// TIA Portal V18 export
FUNCTION_BLOCK "ST10_Flow3_A1RotaryShaftScan"   // FB1073, GRAPH
VERSION : 0.1
// stored: AcknowledgeErrorsRequired false, AutoNumber false, GraphVersion 6.0, InitialValuesAcquisition false, IsIECCheckEnabled false, LanguageInNetworks LAD, LockOperatingMode false, PermanentILProcessingInMANMode false, SetENOAutomatically false, SkipSteps false, UDAEnableTagReadback false, WithAlarmHandling true
   // inherited from GRAPH_BASE
   VAR
      OFF_SQ_BASE : Bool;
   END_VAR
   VAR_INPUT
      iSysInface : "RCS_SysComInterface_V1";
   END_VAR
   VAR_IN_OUT
      ioPM_Inface : "RCS_PMInterface_V1";
      ioStatus : Int;
   END_VAR
   VAR
      sCtrlMode { S7_SetPoint := 'True'} : "SysFlowCtrlGraph";
      sUpdMES_Data : Bool;   // 更新MES数据
      工件放行中 : Bool;
      前站站号 { ExternalAccessible := 'False'; ExternalVisible := 'False'; ExternalWritable := 'False'} : UInt;
      本站站号 { ExternalAccessible := 'False'; ExternalVisible := 'False'; ExternalWritable := 'False'} : UInt;
      弹窗Temp : Array[1..10] of Int;
      AlarmID : Int;
      TON { S7_SetPoint := 'True'} : Array[0..10] of TON_TIME;
      TOF { S7_SetPoint := 'True'} : Array[0..10] of TOF_TIME;
      sUP { S7_SetPoint := 'True'} : Array[0..10] of Bool;
      更新RFID完成 : Bool;
   END_VAR
   VAR_TEMP
      Tempresult : USInt;
      本站站号乘10 : UInt;
   END_VAR
   // // TON[0] : 托盘流入1托盘到位传感器 / iA-Rotating product Check
   // // TON[1] : 托盘流入1托盘到位传感器
   // // TON[2] : 托盘流入1产品有无传感器
   // // TON[3] : 托盘流入1产品有无传感器
   // // TON[4] : 托盘流入1姿态检测光电2
   // // TON[5] : 托盘流入1姿态检测光电3
   // // TON[0].Q : 托盘流入1托盘到位 / iA-Rotating product Check
   // // TON[1].Q : 托盘流入1托盘无
   // // TON[2].Q : 托盘流入1有产品
   // // TON[3].Q : 托盘流入1无产品
   // // TON[4].Q : 托盘流入1姿态检测光电2
   // // TON[5].Q : 托盘流入1姿态检测光电3
   // // TOF[1] : iA-Rotating product Check
BEGIN
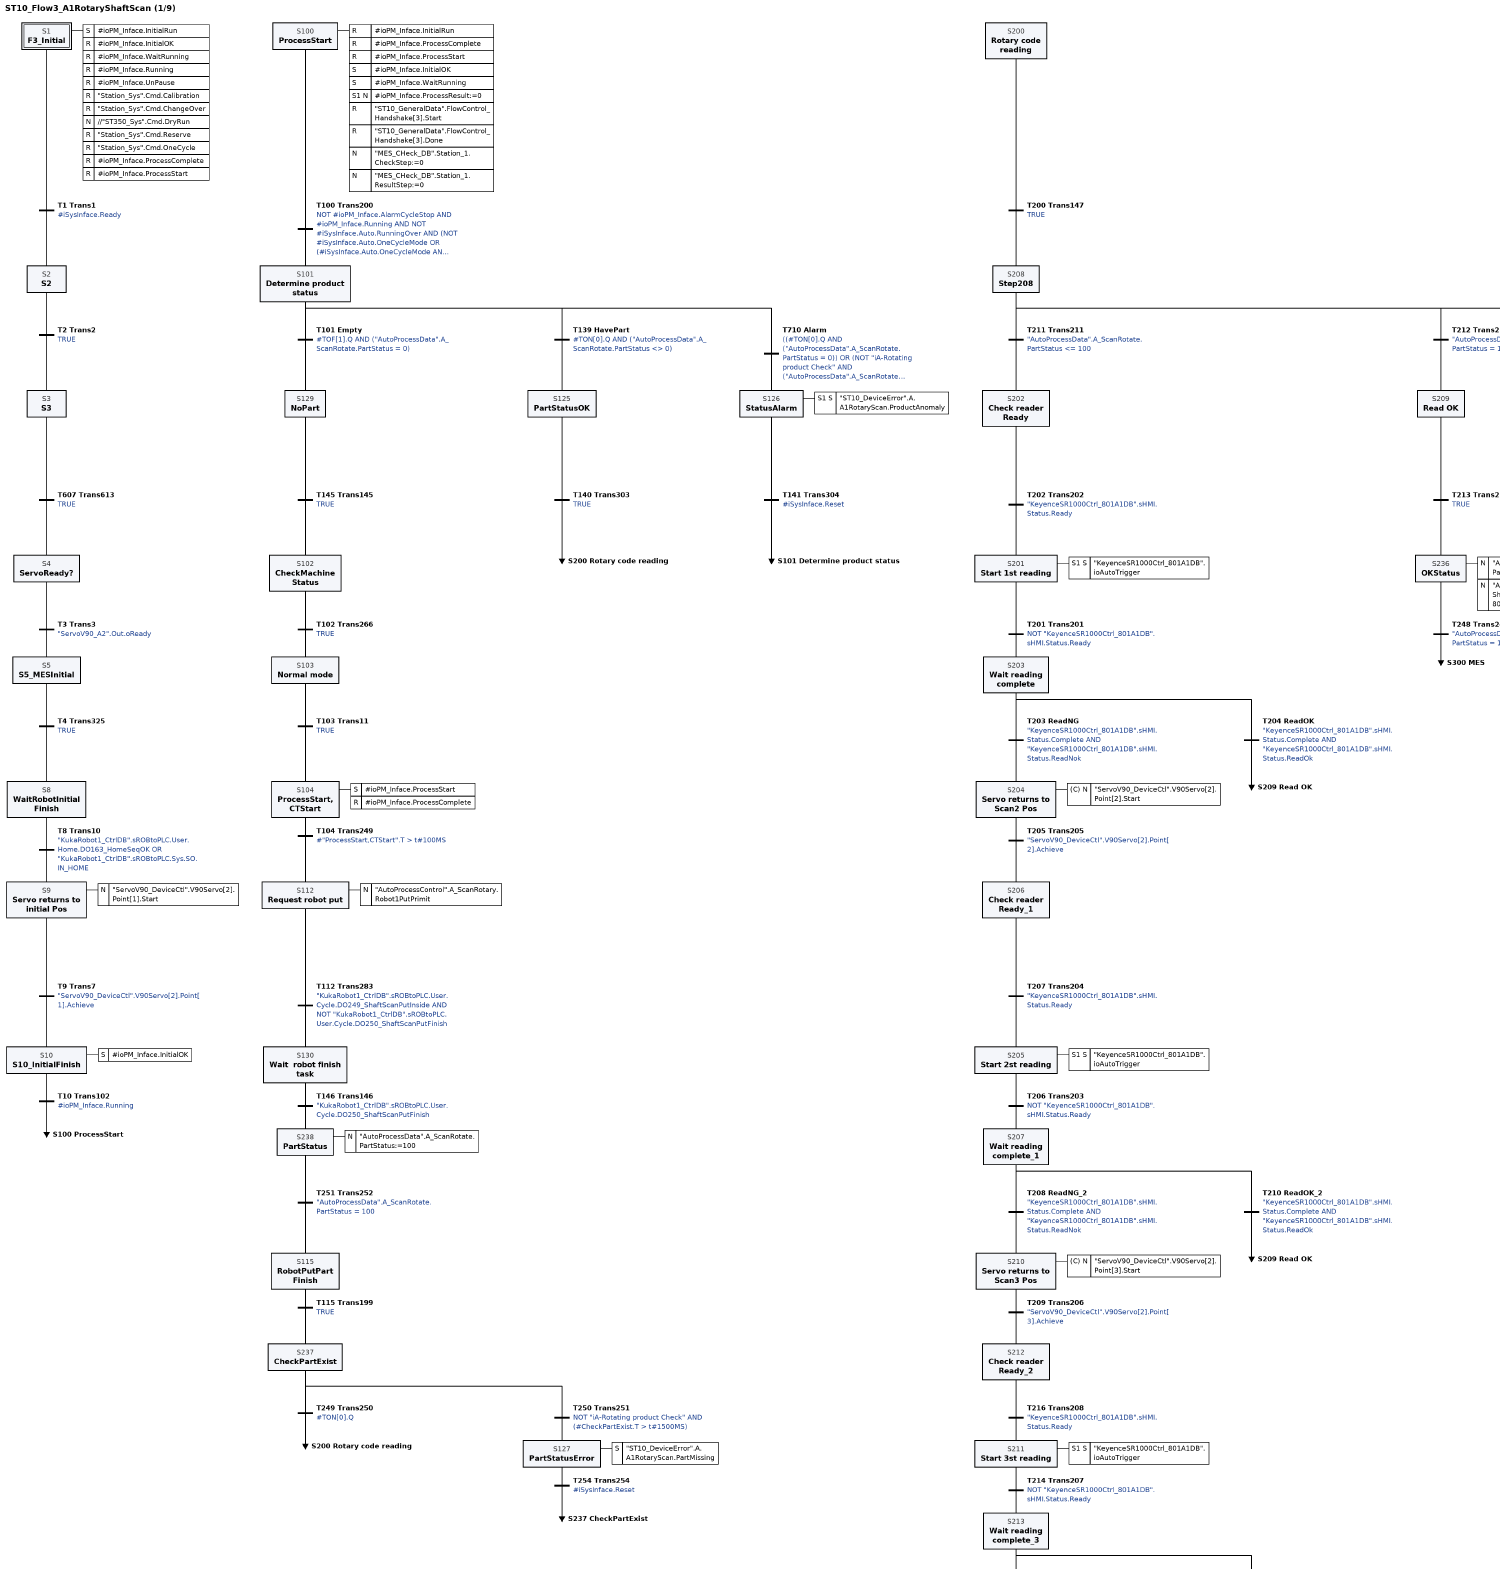
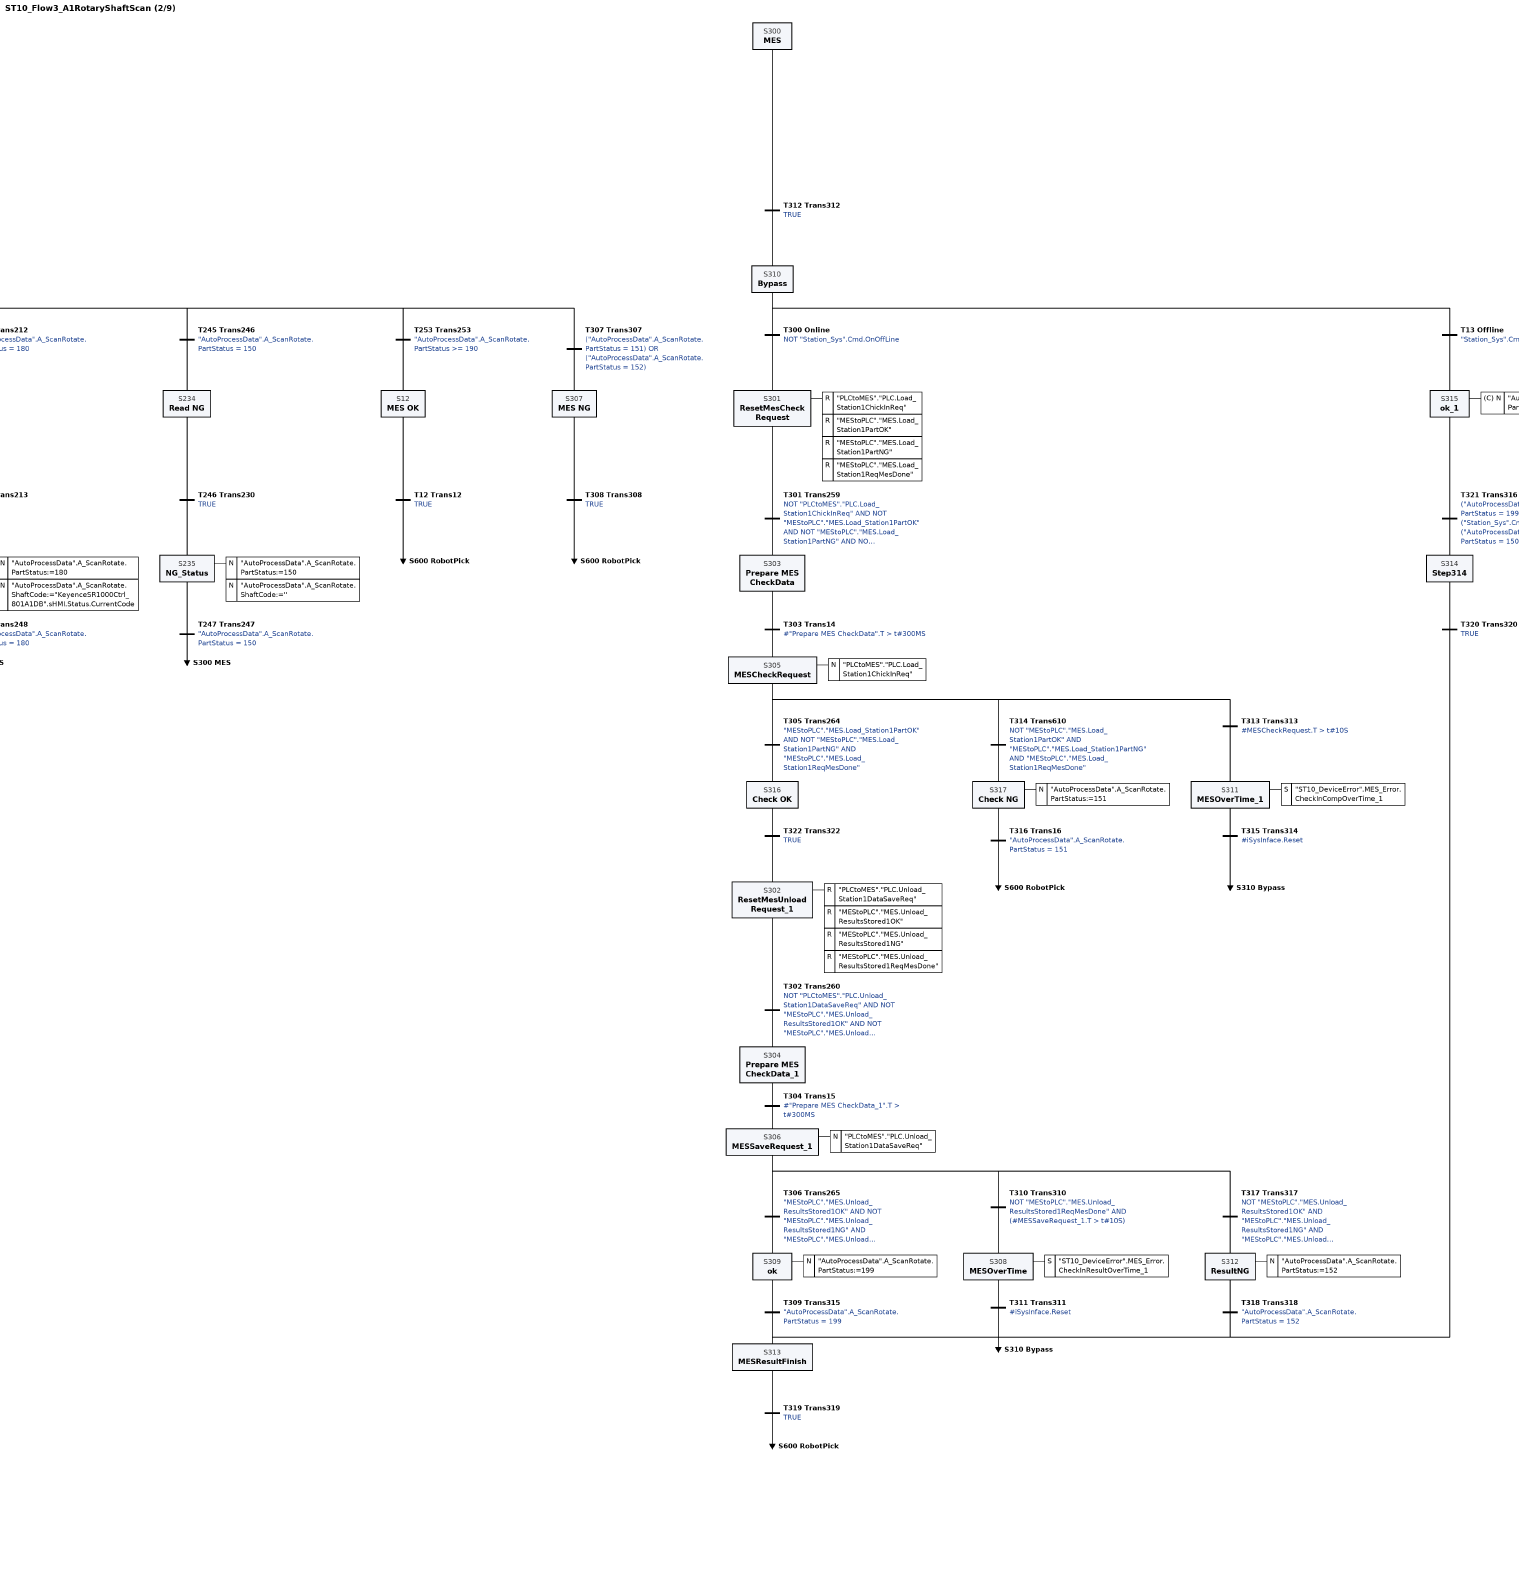
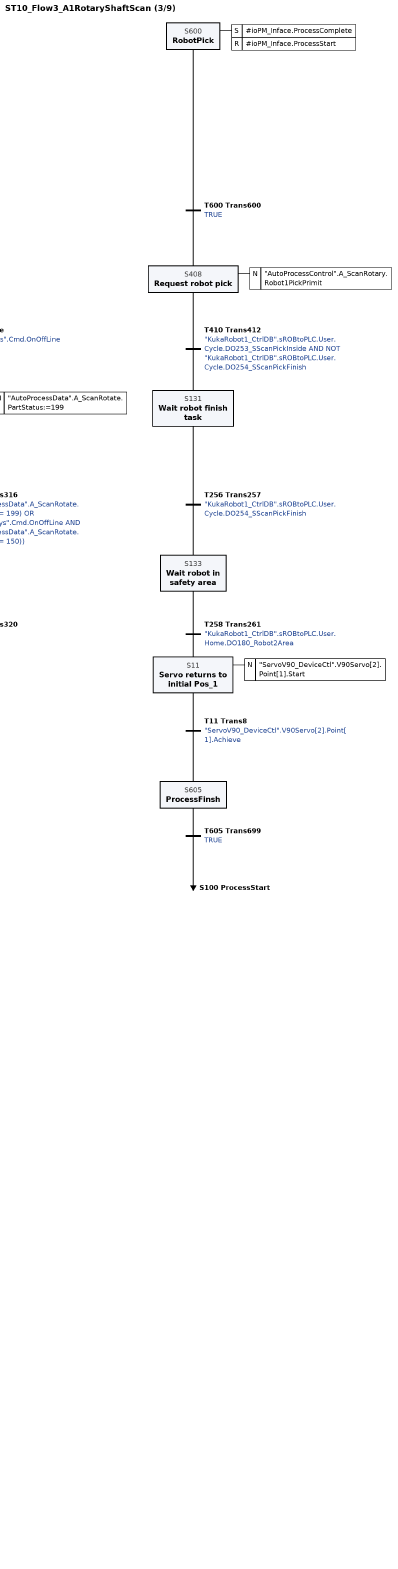
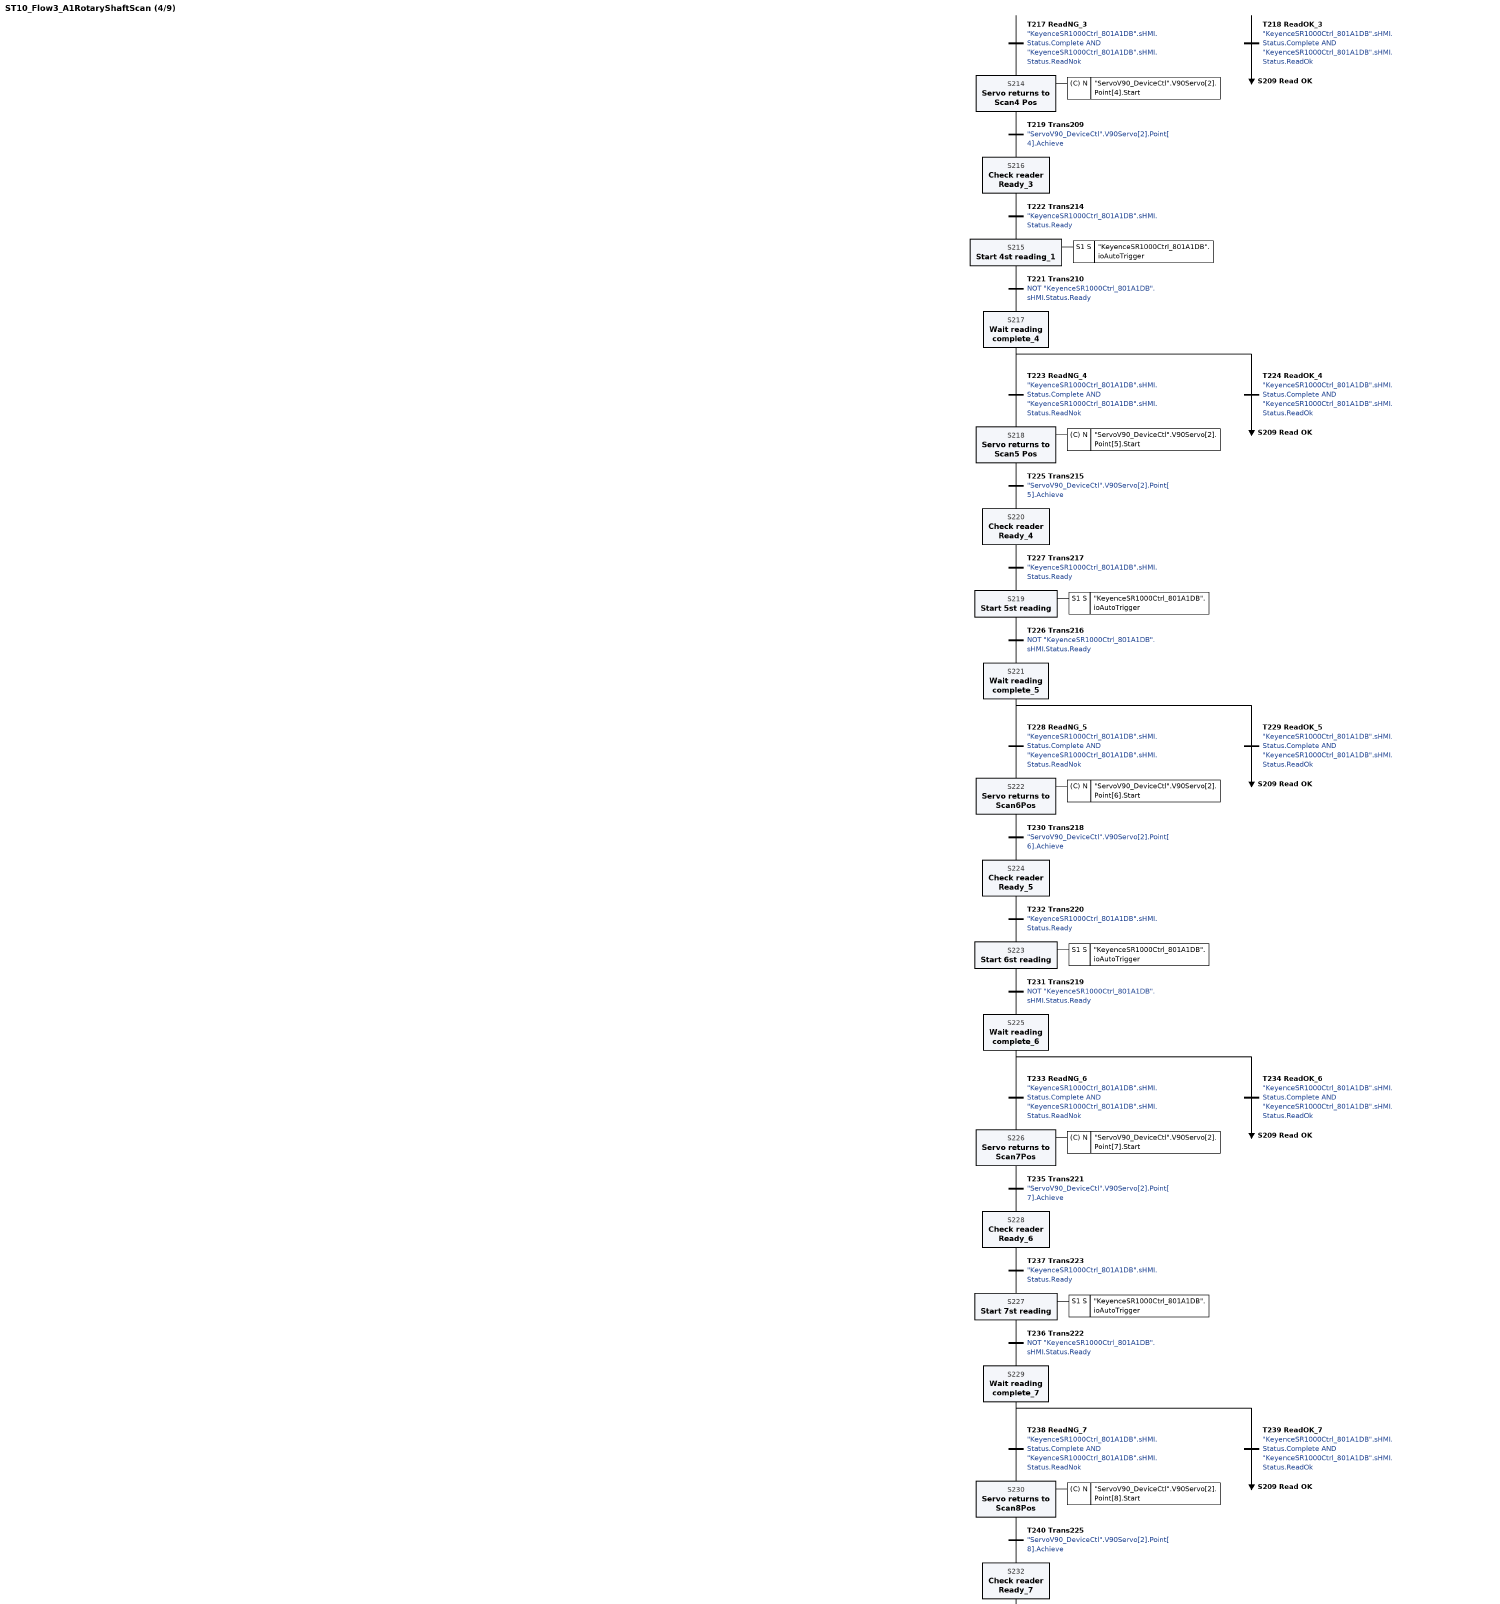
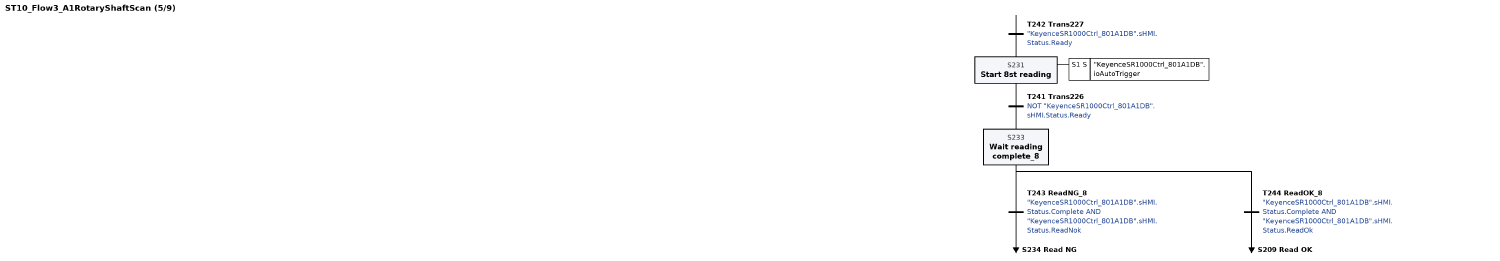
   // permanent pre-instructions
   NETWORK 1
      #TON[10].TON(IN := "AlwaysTRUE" AND "Station_Sys".Alarm.ImmediatelyStop, PT := T#300ms);
      #ioPM_Inface.AlarmImdilyStop := #TON[10].Q;
      #ioPM_Inface.AlarmCycleStop := "AlwaysTRUE" AND "Station_Sys".Alarm.CycleStop;
   NETWORK 2
      IF NOT False THEN
          #sCtrlMode(iSysInface := #iSysInface, ioPM_Inface := #ioPM_Inface, ioGraphCtrl := #RT_DATA.MOP);   // "SysFlowCtrlGraph"
      END_IF;
   NETWORK 3
      #TON[0].TON(IN := "AlwaysTRUE" AND "iA-Rotating product Check", PT := t#500ms);   // 工位11有托盘
      #TOF[1].TOF(IN := "AlwaysTRUE" AND NOT "iA-Rotating product Check", PT := T#300ms);   // 工位无托盘
      #TON[2].TON(IN := "AlwaysTRUE", PT := T#300ms);
      #TON[3].TON(IN := "AlwaysTRUE", PT := T#300ms);
      #TON[4].TON(IN := "AlwaysTRUE", PT := T#300ms);
      #TON[5].TON(IN := "AlwaysTRUE", PT := T#300ms);
   NETWORK 4
      #前站站号 := 345;
      #本站站号 := 350;

   // sequencer 1: S01-S99 初始化 / S01-S99 Initial
   INITIAL_STEP F3_Initial:   // S1, max time T#10S, warning time T#7S
              S    #ioPM_Inface.InitialRun
              R    #ioPM_Inface.InitialOK
              R    #ioPM_Inface.WaitRunning
              R    #ioPM_Inface.Running
              R    #ioPM_Inface.UnPause
              R    "Station_Sys".Cmd.Calibration
              R    "Station_Sys".Cmd.ChangeOver
                   //"ST350_Sys".Cmd.DryRun
              R    "Station_Sys".Cmd.Reserve
              R    "Station_Sys".Cmd.OneCycle
              R    #ioPM_Inface.ProcessComplete
              R    #ioPM_Inface.ProcessStart
   END_STEP
   TRANSITION Trans1 FROM F3_Initial TO S2   // T1
      := #iSysInface.Ready;
   END_TRANSITION
   STEP S2:   // S2, max time T#10S, warning time T#7S
   END_STEP
   TRANSITION Trans2 FROM S2 TO S3   // T2
      := TRUE;
   END_TRANSITION
   STEP "ServoReady?":   // S4, max time T#10S, warning time T#7S
   END_STEP
   TRANSITION Trans3 FROM "ServoReady?" TO S5_MESInitial   // T3
      := "ServoV90_A2".Out.oReady;
   END_TRANSITION
   STEP S5_MESInitial:   // S5, max time T#10S, warning time T#7S
   END_STEP
   TRANSITION Trans325 FROM S5_MESInitial TO WaitRobotInitialFinish   // T4
      := TRUE;
   END_TRANSITION
   STEP S10_InitialFinish:   // S10, max time T#10S, warning time T#7S
              S    #ioPM_Inface.InitialOK
   END_STEP
   TRANSITION Trans102 FROM S10_InitialFinish TO ProcessStart   // T10, jump
      := #ioPM_Inface.Running;
   END_TRANSITION
   STEP S3:   // S3, max time T#10S, warning time T#7S
   END_STEP
   TRANSITION Trans613 FROM S3 TO "ServoReady?"   // T607
      := TRUE;
   END_TRANSITION
   STEP WaitRobotInitialFinish:   // S8, max time T#10S, warning time T#7S
   END_STEP
   TRANSITION Trans10 FROM WaitRobotInitialFinish TO "Servo returns to initial Pos"   // T8
      := "KukaRobot1_CtrlDB".sROBtoPLC.User.Home.DO163_HomeSeqOK OR "KukaRobot1_CtrlDB".sROBtoPLC.Sys.SO.IN_HOME;
   END_TRANSITION
   STEP "Servo returns to initial Pos":   // S9, max time T#10S, warning time T#7S
              N    "ServoV90_DeviceCtl".V90Servo[2].Point[1].Start
   END_STEP
   TRANSITION Trans7 FROM "Servo returns to initial Pos" TO S10_InitialFinish   // T9
      := "ServoV90_DeviceCtl".V90Servo[2].Point[1].Achieve;
   END_TRANSITION

   // sequencer 2: S100-S199 等待到位 / S100-S199 CheckPartStatus
   STEP "Wait  robot finish task":   // S130, max time T#10S, warning time T#7S
   END_STEP
   TRANSITION Trans146 FROM "Wait  robot finish task" TO PartStatus   // T146
      := "KukaRobot1_CtrlDB".sROBtoPLC.User.Cycle.DO250_ShaftScanPutFinish;
   END_TRANSITION
   STEP CheckMachineStatus:   // S102, max time T#10S, warning time T#7S
   END_STEP
   TRANSITION Trans266 FROM CheckMachineStatus TO "Normal mode"   // T102
      := TRUE;
   END_TRANSITION
   STEP "Normal mode":   // S103, max time T#10S, warning time T#7S
   END_STEP
   TRANSITION Trans11 FROM "Normal mode" TO "ProcessStart,CTStart"   // T103
      := TRUE;
   END_TRANSITION
   STEP RobotPutPartFinish:   // S115, max time T#10S, warning time T#7S
   END_STEP
   TRANSITION Trans199 FROM RobotPutPartFinish TO CheckPartExist   // T115
      := TRUE;
   END_TRANSITION
   STEP ProcessStart:   // S100, max time T#10S, warning time T#7S
      // 自动等待开始运行
              R    #ioPM_Inface.InitialRun
              R    #ioPM_Inface.ProcessComplete
              R    #ioPM_Inface.ProcessStart
              S    #ioPM_Inface.InitialOK
              S    #ioPM_Inface.WaitRunning
          S1  N    #ioPM_Inface.ProcessResult:=0
              R    "ST10_GeneralData".FlowControl_Handshake[3].Start
              R    "ST10_GeneralData".FlowControl_Handshake[3].Done
              N    "MES_CHeck_DB".Station_1.CheckStep:=0
              N    "MES_CHeck_DB".Station_1.ResultStep:=0
   END_STEP
   TRANSITION Trans200 FROM ProcessStart TO "Determine product status"   // T100
      := NOT #ioPM_Inface.AlarmCycleStop AND #ioPM_Inface.Running AND NOT #iSysInface.Auto.RunningOver AND (NOT #iSysInface.Auto.OneCycleMode OR (#iSysInface.Auto.OneCycleMode AND #ioPM_Inface.TriggerOneCycle));
   END_TRANSITION
   STEP "ProcessStart,CTStart":   // S104, max time T#10S, warning time T#7S
              S    #ioPM_Inface.ProcessStart
              R    #ioPM_Inface.ProcessComplete
   END_STEP
   TRANSITION Trans249 FROM "ProcessStart,CTStart" TO "Request robot put"   // T104
      := #"ProcessStart,CTStart".T > t#100MS;
   END_TRANSITION
   STEP CheckPartExist:   // S237, max time T#10S, warning time T#7S
   END_STEP
   TRANSITION Trans250 FROM CheckPartExist TO "Rotary code reading"   // T249, jump
      := #TON[0].Q;
   END_TRANSITION
   TRANSITION Trans251 FROM CheckPartExist TO PartStatusError   // T250
      := NOT "iA-Rotating product Check" AND (#CheckPartExist.T > t#1500MS);
   END_TRANSITION
   STEP "Request robot put":   // S112, max time T#10S, warning time T#7S
              N    "AutoProcessControl".A_ScanRotary.Robot1PutPrimit
   END_STEP
   TRANSITION Trans283 FROM "Request robot put" TO "Wait  robot finish task"   // T112
      := "KukaRobot1_CtrlDB".sROBtoPLC.User.Cycle.DO249_ShaftScanPutInside AND NOT "KukaRobot1_CtrlDB".sROBtoPLC.User.Cycle.DO250_ShaftScanPutFinish;
   END_TRANSITION
   STEP PartStatusError:   // S127, max time T#10S, warning time T#7S
              S    "ST10_DeviceError".A.A1RotaryScan.PartMissing
   END_STEP
   TRANSITION Trans254 FROM PartStatusError TO CheckPartExist   // T254, jump
      := #iSysInface.Reset;
   END_TRANSITION
   STEP PartStatus:   // S238, max time T#10S, warning time T#7S
              N    "AutoProcessData".A_ScanRotate.PartStatus:=100
   END_STEP
   TRANSITION Trans252 FROM PartStatus TO RobotPutPartFinish   // T251
      := "AutoProcessData".A_ScanRotate.PartStatus = 100;
   END_TRANSITION
   STEP "Determine product status":   // S101, max time T#10S, warning time T#7S
   END_STEP
   TRANSITION Empty FROM "Determine product status" TO NoPart   // T101
      := #TOF[1].Q AND ("AutoProcessData".A_ScanRotate.PartStatus = 0);
   END_TRANSITION
   TRANSITION HavePart FROM "Determine product status" TO PartStatusOK   // T139
      := #TON[0].Q AND ("AutoProcessData".A_ScanRotate.PartStatus <> 0);
   END_TRANSITION
   TRANSITION Alarm FROM "Determine product status" TO StatusAlarm   // T710
      := ((#TON[0].Q AND ("AutoProcessData".A_ScanRotate.PartStatus = 0)) OR (NOT "iA-Rotating product Check" AND ("AutoProcessData".A_ScanRotate.PartStatus <> 0))) AND (#"Determine product status".T > t#1500MS);
   END_TRANSITION
   STEP PartStatusOK:   // S125, max time T#10S, warning time T#7S
   END_STEP
   TRANSITION Trans303 FROM PartStatusOK TO "Rotary code reading"   // T140, jump
      := TRUE;
   END_TRANSITION
   STEP StatusAlarm:   // S126, max time T#10S, warning time T#7S
          S1  S    "ST10_DeviceError".A.A1RotaryScan.ProductAnomaly
   END_STEP
   TRANSITION Trans304 FROM StatusAlarm TO "Determine product status"   // T141, jump
      := #iSysInface.Reset;
   END_TRANSITION
   STEP NoPart:   // S129, max time T#10S, warning time T#7S
   END_STEP
   TRANSITION Trans145 FROM NoPart TO CheckMachineStatus   // T145
      := TRUE;
   END_TRANSITION

   // sequencer 3: S200-S299Rotary code reading
   STEP "Rotary code reading":   // S200, max time T#10S, warning time T#7S
   END_STEP
   TRANSITION Trans147 FROM "Rotary code reading" TO Step208   // T200
      := TRUE;
   END_TRANSITION
   STEP "Start 1st reading":   // S201, max time T#10S, warning time T#7S
          S1  S    "KeyenceSR1000Ctrl_801A1DB".ioAutoTrigger
   END_STEP
   TRANSITION Trans201 FROM "Start 1st reading" TO "Wait reading complete"   // T201
      := NOT "KeyenceSR1000Ctrl_801A1DB".sHMI.Status.Ready;
   END_TRANSITION
   STEP "Check reader Ready":   // S202, max time T#10S, warning time T#7S
   END_STEP
   TRANSITION Trans202 FROM "Check reader Ready" TO "Start 1st reading"   // T202
      := "KeyenceSR1000Ctrl_801A1DB".sHMI.Status.Ready;
   END_TRANSITION
   STEP "Wait reading complete":   // S203, max time T#10S, warning time T#7S
   END_STEP
   TRANSITION ReadNG FROM "Wait reading complete" TO "Servo returns to Scan2 Pos"   // T203
      := "KeyenceSR1000Ctrl_801A1DB".sHMI.Status.Complete AND "KeyenceSR1000Ctrl_801A1DB".sHMI.Status.ReadNok;
   END_TRANSITION
   TRANSITION ReadOK FROM "Wait reading complete" TO "Read OK"   // T204, jump
      := "KeyenceSR1000Ctrl_801A1DB".sHMI.Status.Complete AND "KeyenceSR1000Ctrl_801A1DB".sHMI.Status.ReadOk;
   END_TRANSITION
   STEP "Servo returns to Scan2 Pos":   // S204, max time T#10S, warning time T#7S
      interlock C := "ServoV90_A2".Out.oReady;
      (C)     N    "ServoV90_DeviceCtl".V90Servo[2].Point[2].Start
   END_STEP
   TRANSITION Trans205 FROM "Servo returns to Scan2 Pos" TO "Check reader Ready_1"   // T205
      := "ServoV90_DeviceCtl".V90Servo[2].Point[2].Achieve;
   END_TRANSITION
   STEP "Start 2st reading":   // S205, max time T#10S, warning time T#7S
          S1  S    "KeyenceSR1000Ctrl_801A1DB".ioAutoTrigger
   END_STEP
   TRANSITION Trans203 FROM "Start 2st reading" TO "Wait reading complete_1"   // T206
      := NOT "KeyenceSR1000Ctrl_801A1DB".sHMI.Status.Ready;
   END_TRANSITION
   STEP "Check reader Ready_1":   // S206, max time T#10S, warning time T#7S
   END_STEP
   TRANSITION Trans204 FROM "Check reader Ready_1" TO "Start 2st reading"   // T207
      := "KeyenceSR1000Ctrl_801A1DB".sHMI.Status.Ready;
   END_TRANSITION
   STEP "Wait reading complete_1":   // S207, max time T#10S, warning time T#7S
   END_STEP
   TRANSITION ReadNG_2 FROM "Wait reading complete_1" TO "Servo returns to Scan3 Pos"   // T208
      := "KeyenceSR1000Ctrl_801A1DB".sHMI.Status.Complete AND "KeyenceSR1000Ctrl_801A1DB".sHMI.Status.ReadNok;
   END_TRANSITION
   TRANSITION ReadOK_2 FROM "Wait reading complete_1" TO "Read OK"   // T210, jump
      := "KeyenceSR1000Ctrl_801A1DB".sHMI.Status.Complete AND "KeyenceSR1000Ctrl_801A1DB".sHMI.Status.ReadOk;
   END_TRANSITION
   STEP Step208:   // S208, max time T#10S, warning time T#7S
   END_STEP
   TRANSITION Trans211 FROM Step208 TO "Check reader Ready"   // T211
      := "AutoProcessData".A_ScanRotate.PartStatus <= 100;
   END_TRANSITION
   TRANSITION Trans212 FROM Step208 TO "Read OK"   // T212
      := "AutoProcessData".A_ScanRotate.PartStatus = 180;
   END_TRANSITION
   TRANSITION Trans246 FROM Step208 TO "Read NG"   // T245
      := "AutoProcessData".A_ScanRotate.PartStatus = 150;
   END_TRANSITION
   TRANSITION Trans253 FROM Step208 TO "MES OK"   // T253
      := "AutoProcessData".A_ScanRotate.PartStatus >= 190;
   END_TRANSITION
   TRANSITION Trans307 FROM Step208 TO "MES NG"   // T307
      := ("AutoProcessData".A_ScanRotate.PartStatus = 151) OR ("AutoProcessData".A_ScanRotate.PartStatus = 152);
   END_TRANSITION
   STEP "Read OK":   // S209, max time T#10S, warning time T#7S
   END_STEP
   TRANSITION Trans213 FROM "Read OK" TO OKStatus   // T213
      := TRUE;
   END_TRANSITION
   STEP "Servo returns to Scan3 Pos":   // S210, max time T#10S, warning time T#7S
      interlock C := "ServoV90_A2".Out.oReady;
      (C)     N    "ServoV90_DeviceCtl".V90Servo[2].Point[3].Start
   END_STEP
   TRANSITION Trans206 FROM "Servo returns to Scan3 Pos" TO "Check reader Ready_2"   // T209
      := "ServoV90_DeviceCtl".V90Servo[2].Point[3].Achieve;
   END_TRANSITION
   STEP "Start 3st reading":   // S211, max time T#10S, warning time T#7S
          S1  S    "KeyenceSR1000Ctrl_801A1DB".ioAutoTrigger
   END_STEP
   TRANSITION Trans207 FROM "Start 3st reading" TO "Wait reading complete_3"   // T214
      := NOT "KeyenceSR1000Ctrl_801A1DB".sHMI.Status.Ready;
   END_TRANSITION
   STEP "Check reader Ready_2":   // S212, max time T#10S, warning time T#7S
   END_STEP
   TRANSITION Trans208 FROM "Check reader Ready_2" TO "Start 3st reading"   // T216
      := "KeyenceSR1000Ctrl_801A1DB".sHMI.Status.Ready;
   END_TRANSITION
   STEP "Wait reading complete_3":   // S213, max time T#10S, warning time T#7S
   END_STEP
   TRANSITION ReadNG_3 FROM "Wait reading complete_3" TO "Servo returns to Scan4 Pos"   // T217
      := "KeyenceSR1000Ctrl_801A1DB".sHMI.Status.Complete AND "KeyenceSR1000Ctrl_801A1DB".sHMI.Status.ReadNok;
   END_TRANSITION
   TRANSITION ReadOK_3 FROM "Wait reading complete_3" TO "Read OK"   // T218, jump
      := "KeyenceSR1000Ctrl_801A1DB".sHMI.Status.Complete AND "KeyenceSR1000Ctrl_801A1DB".sHMI.Status.ReadOk;
   END_TRANSITION
   STEP "Servo returns to Scan4 Pos":   // S214, max time T#10S, warning time T#7S
      interlock C := "ServoV90_A2".Out.oReady;
      (C)     N    "ServoV90_DeviceCtl".V90Servo[2].Point[4].Start
   END_STEP
   TRANSITION Trans209 FROM "Servo returns to Scan4 Pos" TO "Check reader Ready_3"   // T219
      := "ServoV90_DeviceCtl".V90Servo[2].Point[4].Achieve;
   END_TRANSITION
   STEP "Start 4st reading_1":   // S215, max time T#10S, warning time T#7S
          S1  S    "KeyenceSR1000Ctrl_801A1DB".ioAutoTrigger
   END_STEP
   TRANSITION Trans210 FROM "Start 4st reading_1" TO "Wait reading complete_4"   // T221
      := NOT "KeyenceSR1000Ctrl_801A1DB".sHMI.Status.Ready;
   END_TRANSITION
   STEP "Check reader Ready_3":   // S216, max time T#10S, warning time T#7S
   END_STEP
   TRANSITION Trans214 FROM "Check reader Ready_3" TO "Start 4st reading_1"   // T222
      := "KeyenceSR1000Ctrl_801A1DB".sHMI.Status.Ready;
   END_TRANSITION
   STEP "Wait reading complete_4":   // S217, max time T#10S, warning time T#7S
   END_STEP
   TRANSITION ReadNG_4 FROM "Wait reading complete_4" TO "Servo returns to Scan5 Pos"   // T223
      := "KeyenceSR1000Ctrl_801A1DB".sHMI.Status.Complete AND "KeyenceSR1000Ctrl_801A1DB".sHMI.Status.ReadNok;
   END_TRANSITION
   TRANSITION ReadOK_4 FROM "Wait reading complete_4" TO "Read OK"   // T224, jump
      := "KeyenceSR1000Ctrl_801A1DB".sHMI.Status.Complete AND "KeyenceSR1000Ctrl_801A1DB".sHMI.Status.ReadOk;
   END_TRANSITION
   STEP "Servo returns to Scan5 Pos":   // S218, max time T#10S, warning time T#7S
      interlock C := "ServoV90_A2".Out.oReady;
      (C)     N    "ServoV90_DeviceCtl".V90Servo[2].Point[5].Start
   END_STEP
   TRANSITION Trans215 FROM "Servo returns to Scan5 Pos" TO "Check reader Ready_4"   // T225
      := "ServoV90_DeviceCtl".V90Servo[2].Point[5].Achieve;
   END_TRANSITION
   STEP "Start 5st reading":   // S219, max time T#10S, warning time T#7S
          S1  S    "KeyenceSR1000Ctrl_801A1DB".ioAutoTrigger
   END_STEP
   TRANSITION Trans216 FROM "Start 5st reading" TO "Wait reading complete_5"   // T226
      := NOT "KeyenceSR1000Ctrl_801A1DB".sHMI.Status.Ready;
   END_TRANSITION
   STEP "Check reader Ready_4":   // S220, max time T#10S, warning time T#7S
   END_STEP
   TRANSITION Trans217 FROM "Check reader Ready_4" TO "Start 5st reading"   // T227
      := "KeyenceSR1000Ctrl_801A1DB".sHMI.Status.Ready;
   END_TRANSITION
   STEP "Wait reading complete_5":   // S221, max time T#10S, warning time T#7S
   END_STEP
   TRANSITION ReadNG_5 FROM "Wait reading complete_5" TO "Servo returns to Scan6Pos"   // T228
      := "KeyenceSR1000Ctrl_801A1DB".sHMI.Status.Complete AND "KeyenceSR1000Ctrl_801A1DB".sHMI.Status.ReadNok;
   END_TRANSITION
   TRANSITION ReadOK_5 FROM "Wait reading complete_5" TO "Read OK"   // T229, jump
      := "KeyenceSR1000Ctrl_801A1DB".sHMI.Status.Complete AND "KeyenceSR1000Ctrl_801A1DB".sHMI.Status.ReadOk;
   END_TRANSITION
   STEP "Servo returns to Scan6Pos":   // S222, max time T#10S, warning time T#7S
      interlock C := "ServoV90_A2".Out.oReady;
      (C)     N    "ServoV90_DeviceCtl".V90Servo[2].Point[6].Start
   END_STEP
   TRANSITION Trans218 FROM "Servo returns to Scan6Pos" TO "Check reader Ready_5"   // T230
      := "ServoV90_DeviceCtl".V90Servo[2].Point[6].Achieve;
   END_TRANSITION
   STEP "Start 6st reading":   // S223, max time T#10S, warning time T#7S
          S1  S    "KeyenceSR1000Ctrl_801A1DB".ioAutoTrigger
   END_STEP
   TRANSITION Trans219 FROM "Start 6st reading" TO "Wait reading complete_6"   // T231
      := NOT "KeyenceSR1000Ctrl_801A1DB".sHMI.Status.Ready;
   END_TRANSITION
   STEP "Check reader Ready_5":   // S224, max time T#10S, warning time T#7S
   END_STEP
   TRANSITION Trans220 FROM "Check reader Ready_5" TO "Start 6st reading"   // T232
      := "KeyenceSR1000Ctrl_801A1DB".sHMI.Status.Ready;
   END_TRANSITION
   STEP "Wait reading complete_6":   // S225, max time T#10S, warning time T#7S
   END_STEP
   TRANSITION ReadNG_6 FROM "Wait reading complete_6" TO "Servo returns to Scan7Pos"   // T233
      := "KeyenceSR1000Ctrl_801A1DB".sHMI.Status.Complete AND "KeyenceSR1000Ctrl_801A1DB".sHMI.Status.ReadNok;
   END_TRANSITION
   TRANSITION ReadOK_6 FROM "Wait reading complete_6" TO "Read OK"   // T234, jump
      := "KeyenceSR1000Ctrl_801A1DB".sHMI.Status.Complete AND "KeyenceSR1000Ctrl_801A1DB".sHMI.Status.ReadOk;
   END_TRANSITION
   STEP "Servo returns to Scan7Pos":   // S226, max time T#10S, warning time T#7S
      interlock C := "ServoV90_A2".Out.oReady;
      (C)     N    "ServoV90_DeviceCtl".V90Servo[2].Point[7].Start
   END_STEP
   TRANSITION Trans221 FROM "Servo returns to Scan7Pos" TO "Check reader Ready_6"   // T235
      := "ServoV90_DeviceCtl".V90Servo[2].Point[7].Achieve;
   END_TRANSITION
   STEP "Start 7st reading":   // S227, max time T#10S, warning time T#7S
          S1  S    "KeyenceSR1000Ctrl_801A1DB".ioAutoTrigger
   END_STEP
   TRANSITION Trans222 FROM "Start 7st reading" TO "Wait reading complete_7"   // T236
      := NOT "KeyenceSR1000Ctrl_801A1DB".sHMI.Status.Ready;
   END_TRANSITION
   STEP "Check reader Ready_6":   // S228, max time T#10S, warning time T#7S
   END_STEP
   TRANSITION Trans223 FROM "Check reader Ready_6" TO "Start 7st reading"   // T237
      := "KeyenceSR1000Ctrl_801A1DB".sHMI.Status.Ready;
   END_TRANSITION
   STEP "Wait reading complete_7":   // S229, max time T#10S, warning time T#7S
   END_STEP
   TRANSITION ReadNG_7 FROM "Wait reading complete_7" TO "Servo returns to Scan8Pos"   // T238
      := "KeyenceSR1000Ctrl_801A1DB".sHMI.Status.Complete AND "KeyenceSR1000Ctrl_801A1DB".sHMI.Status.ReadNok;
   END_TRANSITION
   TRANSITION ReadOK_7 FROM "Wait reading complete_7" TO "Read OK"   // T239, jump
      := "KeyenceSR1000Ctrl_801A1DB".sHMI.Status.Complete AND "KeyenceSR1000Ctrl_801A1DB".sHMI.Status.ReadOk;
   END_TRANSITION
   STEP "Servo returns to Scan8Pos":   // S230, max time T#10S, warning time T#7S
      interlock C := "ServoV90_A2".Out.oReady;
      (C)     N    "ServoV90_DeviceCtl".V90Servo[2].Point[8].Start
   END_STEP
   TRANSITION Trans225 FROM "Servo returns to Scan8Pos" TO "Check reader Ready_7"   // T240
      := "ServoV90_DeviceCtl".V90Servo[2].Point[8].Achieve;
   END_TRANSITION
   STEP "Start 8st reading":   // S231, max time T#10S, warning time T#7S
          S1  S    "KeyenceSR1000Ctrl_801A1DB".ioAutoTrigger
   END_STEP
   TRANSITION Trans226 FROM "Start 8st reading" TO "Wait reading complete_8"   // T241
      := NOT "KeyenceSR1000Ctrl_801A1DB".sHMI.Status.Ready;
   END_TRANSITION
   STEP "Check reader Ready_7":   // S232, max time T#10S, warning time T#7S
   END_STEP
   TRANSITION Trans227 FROM "Check reader Ready_7" TO "Start 8st reading"   // T242
      := "KeyenceSR1000Ctrl_801A1DB".sHMI.Status.Ready;
   END_TRANSITION
   STEP "Wait reading complete_8":   // S233, max time T#10S, warning time T#7S
   END_STEP
   TRANSITION ReadNG_8 FROM "Wait reading complete_8" TO "Read NG"   // T243, jump
      := "KeyenceSR1000Ctrl_801A1DB".sHMI.Status.Complete AND "KeyenceSR1000Ctrl_801A1DB".sHMI.Status.ReadNok;
   END_TRANSITION
   TRANSITION ReadOK_8 FROM "Wait reading complete_8" TO "Read OK"   // T244, jump
      := "KeyenceSR1000Ctrl_801A1DB".sHMI.Status.Complete AND "KeyenceSR1000Ctrl_801A1DB".sHMI.Status.ReadOk;
   END_TRANSITION
   STEP "Read NG":   // S234, max time T#10S, warning time T#7S
   END_STEP
   TRANSITION Trans230 FROM "Read NG" TO NG_Status   // T246
      := TRUE;
   END_TRANSITION
   STEP NG_Status:   // S235, max time T#10S, warning time T#7S
              N    "AutoProcessData".A_ScanRotate.PartStatus:=150
              N    "AutoProcessData".A_ScanRotate.ShaftCode:=''
   END_STEP
   TRANSITION Trans247 FROM NG_Status TO MES   // T247, jump
      := "AutoProcessData".A_ScanRotate.PartStatus = 150;
   END_TRANSITION
   STEP OKStatus:   // S236, max time T#10S, warning time T#7S
              N    "AutoProcessData".A_ScanRotate.PartStatus:=180
              N    "AutoProcessData".A_ScanRotate.ShaftCode:="KeyenceSR1000Ctrl_801A1DB".sHMI.Status.CurrentCode
   END_STEP
   TRANSITION Trans248 FROM OKStatus TO MES   // T248, jump
      := "AutoProcessData".A_ScanRotate.PartStatus = 180;
   END_TRANSITION
   STEP "MES NG":   // S307, max time T#10S, warning time T#7S
   END_STEP
   TRANSITION Trans308 FROM "MES NG" TO RobotPick   // T308, jump
      := TRUE;
   END_TRANSITION
   STEP "MES OK":   // S12, max time T#10S, warning time T#7S
   END_STEP
   TRANSITION Trans12 FROM "MES OK" TO RobotPick   // T12, jump
      := TRUE;
   END_TRANSITION

   // sequencer 4: S200-S299MES查询获取打标数据 / S300-S399 MES
   STEP "Prepare MES CheckData":   // S303, max time T#10S, warning time T#7S
   END_STEP
   TRANSITION Trans14 FROM "Prepare MES CheckData" TO MESCheckRequest   // T303
      := #"Prepare MES CheckData".T > t#300MS;
   END_TRANSITION
   STEP MESCheckRequest:   // S305, max time T#10S, warning time T#7S
              N    "PLCtoMES"."PLC.Load_Station1ChickInReq"
   END_STEP
   TRANSITION Trans264 FROM MESCheckRequest TO "Check OK"   // T305
      := "MEStoPLC"."MES.Load_Station1PartOK" AND NOT "MEStoPLC"."MES.Load_Station1PartNG" AND "MEStoPLC"."MES.Load_Station1ReqMesDone";
   END_TRANSITION
   TRANSITION Trans610 FROM MESCheckRequest TO "Check NG"   // T314
      := NOT "MEStoPLC"."MES.Load_Station1PartOK" AND "MEStoPLC"."MES.Load_Station1PartNG" AND "MEStoPLC"."MES.Load_Station1ReqMesDone";
   END_TRANSITION
   TRANSITION Trans313 FROM MESCheckRequest TO MESOverTime_1   // T313
      := #MESCheckRequest.T > t#10S;
   END_TRANSITION
   STEP MES:   // S300, max time T#10S, warning time T#7S
   END_STEP
   TRANSITION Trans312 FROM MES TO Bypass   // T312
      := TRUE;
   END_TRANSITION
   STEP ResetMesCheckRequest:   // S301, max time T#10S, warning time T#7S
              R    "PLCtoMES"."PLC.Load_Station1ChickInReq"
              R    "MEStoPLC"."MES.Load_Station1PartOK"
              R    "MEStoPLC"."MES.Load_Station1PartNG"
              R    "MEStoPLC"."MES.Load_Station1ReqMesDone"
   END_STEP
   TRANSITION Trans259 FROM ResetMesCheckRequest TO "Prepare MES CheckData"   // T301
      := NOT "PLCtoMES"."PLC.Load_Station1ChickInReq" AND NOT "MEStoPLC"."MES.Load_Station1PartOK" AND NOT "MEStoPLC"."MES.Load_Station1PartNG" AND NOT "MEStoPLC"."MES.Load_Station1ReqMesDone";
   END_TRANSITION
   STEP ok:   // S309, max time T#10S, warning time T#7S
              N    "AutoProcessData".A_ScanRotate.PartStatus:=199
   END_STEP
   TRANSITION Trans315 FROM ok TO MESResultFinish   // T309
      := "AutoProcessData".A_ScanRotate.PartStatus = 199;
   END_TRANSITION
   STEP "Check OK":   // S316, max time T#10S, warning time T#7S
   END_STEP
   TRANSITION Trans322 FROM "Check OK" TO ResetMesUnloadRequest_1   // T322
      := TRUE;
   END_TRANSITION
   STEP "Check NG":   // S317, max time T#10S, warning time T#7S
              N    "AutoProcessData".A_ScanRotate.PartStatus:=151
   END_STEP
   TRANSITION Trans16 FROM "Check NG" TO RobotPick   // T316, jump
      := "AutoProcessData".A_ScanRotate.PartStatus = 151;
   END_TRANSITION
   STEP "Prepare MES CheckData_1":   // S304, max time T#10S, warning time T#7S
   END_STEP
   TRANSITION Trans15 FROM "Prepare MES CheckData_1" TO MESSaveRequest_1   // T304
      := #"Prepare MES CheckData_1".T > t#300MS;
   END_TRANSITION
   STEP MESSaveRequest_1:   // S306, max time T#10S, warning time T#7S
              N    "PLCtoMES"."PLC.Unload_Station1DataSaveReq"
   END_STEP
   TRANSITION Trans265 FROM MESSaveRequest_1 TO ok   // T306
      := "MEStoPLC"."MES.Unload_ResultsStored1OK" AND NOT "MEStoPLC"."MES.Unload_ResultsStored1NG" AND "MEStoPLC"."MES.Unload_ResultsStored1ReqMesDone";
   END_TRANSITION
   TRANSITION Trans310 FROM MESSaveRequest_1 TO MESOverTime   // T310
      := NOT "MEStoPLC"."MES.Unload_ResultsStored1ReqMesDone" AND (#MESSaveRequest_1.T > t#10S);
   END_TRANSITION
   TRANSITION Trans317 FROM MESSaveRequest_1 TO ResultNG   // T317
      := NOT "MEStoPLC"."MES.Unload_ResultsStored1OK" AND "MEStoPLC"."MES.Unload_ResultsStored1NG" AND "MEStoPLC"."MES.Unload_ResultsStored1ReqMesDone";
   END_TRANSITION
   STEP ResetMesUnloadRequest_1:   // S302, max time T#10S, warning time T#7S
              R    "PLCtoMES"."PLC.Unload_Station1DataSaveReq"
              R    "MEStoPLC"."MES.Unload_ResultsStored1OK"
              R    "MEStoPLC"."MES.Unload_ResultsStored1NG"
              R    "MEStoPLC"."MES.Unload_ResultsStored1ReqMesDone"
   END_STEP
   TRANSITION Trans260 FROM ResetMesUnloadRequest_1 TO "Prepare MES CheckData_1"   // T302
      := NOT "PLCtoMES"."PLC.Unload_Station1DataSaveReq" AND NOT "MEStoPLC"."MES.Unload_ResultsStored1OK" AND NOT "MEStoPLC"."MES.Unload_ResultsStored1NG" AND NOT "MEStoPLC"."MES.Unload_ResultsStored1ReqMesDone";
   END_TRANSITION
   STEP MESOverTime:   // S308, max time T#10S, warning time T#7S
              S    "ST10_DeviceError".MES_Error.CheckInResultOverTime_1
   END_STEP
   TRANSITION Trans311 FROM MESOverTime TO Bypass   // T311, jump
      := #iSysInface.Reset;
   END_TRANSITION
   STEP Bypass:   // S310, max time T#10S, warning time T#7S
   END_STEP
   TRANSITION Online FROM Bypass TO ResetMesCheckRequest   // T300
      := NOT "Station_Sys".Cmd.OnOffLine;
   END_TRANSITION
   TRANSITION Offline FROM Bypass TO ok_1   // T13
      := "Station_Sys".Cmd.OnOffLine;
   END_TRANSITION
   STEP MESOverTime_1:   // S311, max time T#10S, warning time T#7S
              S    "ST10_DeviceError".MES_Error.CheckInCompOverTime_1
   END_STEP
   TRANSITION Trans314 FROM MESOverTime_1 TO Bypass   // T315, jump
      := #iSysInface.Reset;
   END_TRANSITION
   STEP ResultNG:   // S312, max time T#10S, warning time T#7S
              N    "AutoProcessData".A_ScanRotate.PartStatus:=152
   END_STEP
   TRANSITION Trans318 FROM ResultNG TO MESResultFinish   // T318
      := "AutoProcessData".A_ScanRotate.PartStatus = 152;
   END_TRANSITION
   STEP MESResultFinish:   // S313, max time T#10S, warning time T#7S
   END_STEP
   TRANSITION Trans319 FROM MESResultFinish TO RobotPick   // T319, jump
      := TRUE;
   END_TRANSITION
   STEP Step314:   // S314, max time T#10S, warning time T#7S
   END_STEP
   TRANSITION Trans320 FROM Step314 TO MESResultFinish   // T320
      := TRUE;
   END_TRANSITION
   STEP ok_1:   // S315, max time T#10S, warning time T#7S
      interlock C := "AutoProcessData".A_ScanRotate.PartStatus = 180;
      (C)     N    "AutoProcessData".A_ScanRotate.PartStatus:=199
   END_STEP
   TRANSITION Trans316 FROM ok_1 TO Step314   // T321
      := ("AutoProcessData".A_ScanRotate.PartStatus = 199) OR ("Station_Sys".Cmd.OnOffLine AND ("AutoProcessData".A_ScanRotate.PartStatus = 150));
   END_TRANSITION

   // sequencer 5: S600-S699工件放行 / S600-S699 RobotPick
   STEP RobotPick:   // S600, max time T#10S, warning time T#7S
              S    #ioPM_Inface.ProcessComplete
              R    #ioPM_Inface.ProcessStart
   END_STEP
   TRANSITION Trans600 FROM RobotPick TO "Request robot pick"   // T600
      := TRUE;
   END_TRANSITION
   STEP ProcessFinsh:   // S605, max time T#10S, warning time T#7S: 正式使用时，需要激活复位空循环
   END_STEP
   TRANSITION Trans699 FROM ProcessFinsh TO ProcessStart   // T605, jump
      := TRUE;
   END_TRANSITION
   STEP "Request robot pick":   // S408, max time T#10S, warning time T#7S
              N    "AutoProcessControl".A_ScanRotary.Robot1PickPrimit
   END_STEP
   TRANSITION Trans412 FROM "Request robot pick" TO "Wait robot finish task"   // T410
      := "KukaRobot1_CtrlDB".sROBtoPLC.User.Cycle.DO253_SScanPickInside AND NOT "KukaRobot1_CtrlDB".sROBtoPLC.User.Cycle.DO254_SScanPickFinish;
   END_TRANSITION
   STEP "Wait robot finish task":   // S131, max time T#10S, warning time T#7S
   END_STEP
   TRANSITION Trans257 FROM "Wait robot finish task" TO "Wait robot in safety area"   // T256
      := "KukaRobot1_CtrlDB".sROBtoPLC.User.Cycle.DO254_SScanPickFinish;
   END_TRANSITION
   STEP "Wait robot in safety area":   // S133, max time T#10S, warning time T#7S
   END_STEP
   TRANSITION Trans261 FROM "Wait robot in safety area" TO "Servo returns to initial Pos_1"   // T258
      := "KukaRobot1_CtrlDB".sROBtoPLC.User.Home.DO180_Robot2Area;
   END_TRANSITION
   STEP "Servo returns to initial Pos_1":   // S11, max time T#10S, warning time T#7S
              N    "ServoV90_DeviceCtl".V90Servo[2].Point[1].Start
   END_STEP
   TRANSITION Trans8 FROM "Servo returns to initial Pos_1" TO ProcessFinsh   // T11
      := "ServoV90_DeviceCtl".V90Servo[2].Point[1].Achieve;
   END_TRANSITION

   // permanent post-instructions
   NETWORK 1
      #ioPM_Inface.StepNum := #RT_DATA.S_DISPLAY;
   NETWORK 2
      IF #iSysInface.Reset THEN #AlarmID := 0; END_IF;
   NETWORK 3
      #TON[10].TON(IN := #工件放行中, PT := T#0.5S);
      IF #TON[10].Q THEN #工件放行中 := FALSE; END_IF;
END_FUNCTION_BLOCK
